// TIA Portal project "Industrial Oven Control" (V17)
// Industrial Oven Control
// The oven should preheat for 10s, then maintain the set temperature for 20 sec and then cool down for 30 sec.

(* hardware
DEVICE "S7-1200 station_1"  S7-1200 Station
   slot 0: "Rack_0"  S7-1200 Rack  Rack  V1.0
   slot 1: "PLC_1"  CPU 1215C AC/DC/Rly  6ES7 215-1BG40-0XB0  V4.5
*)

// ===== PLC "PLC_1"  CPU 1215C AC/DC/Rly =====

VAR_GLOBAL   // PLC tag table "Default tag table"
   "Turn_ON" AT %I0.0 : Bool;
   "Pre-Heat" AT %Q0.0 : Bool;
   "Set Temp" AT %Q0.1 : Bool;
   "Cooling" AT %Q0.2 : Bool;
END_VAR

// folder: System blocks/Program resources

DATA_BLOCK "IEC_Timer_0_DB"   // DB1
{ S7_Optimized_Access := 'TRUE' }
AUTHOR : Simatic
FAMILY : IEC
NAME : IEC_TMR
VERSION : 1.0
// stored: InstanceOfName IEC_TIMER
"IEC_TIMER"
BEGIN
END_DATA_BLOCK

DATA_BLOCK "IEC_Timer_0_DB_1"   // DB2
{ S7_Optimized_Access := 'TRUE' }
AUTHOR : Simatic
FAMILY : IEC
NAME : IEC_TMR
VERSION : 1.0
// stored: InstanceOfName IEC_TIMER
"IEC_TIMER"
BEGIN
END_DATA_BLOCK

DATA_BLOCK "IEC_Timer_0_DB_2"   // DB3
{ S7_Optimized_Access := 'TRUE' }
AUTHOR : Simatic
FAMILY : IEC
NAME : IEC_TMR
VERSION : 1.0
// stored: InstanceOfName IEC_TIMER
"IEC_TIMER"
BEGIN
END_DATA_BLOCK

DATA_BLOCK "IEC_Timer_0_DB_3"   // DB4
{ S7_Optimized_Access := 'TRUE' }
AUTHOR : Simatic
FAMILY : IEC
NAME : IEC_TMR
VERSION : 1.0
// stored: InstanceOfName IEC_TIMER
"IEC_TIMER"
BEGIN
END_DATA_BLOCK

DATA_BLOCK "IEC_Timer_0_DB_4"   // DB5
{ S7_Optimized_Access := 'TRUE' }
AUTHOR : Simatic
FAMILY : IEC
NAME : IEC_TMR
VERSION : 1.0
// stored: InstanceOfName IEC_TIMER
"IEC_TIMER"
BEGIN
END_DATA_BLOCK

// folder: (top level)

ORGANIZATION_BLOCK "Main"   // OB1, LAD, ProgramCycle
TITLE = "Main Program Sweep (Cycle)"
{ S7_Optimized_Access := 'TRUE' }
VERSION : 0.1
   VAR_INPUT
      Initial_Call : Bool;   // Initial call of this OB
      Remanence : Bool;   // =True, if remanent data are available
   END_VAR
BEGIN

REGION Network 1
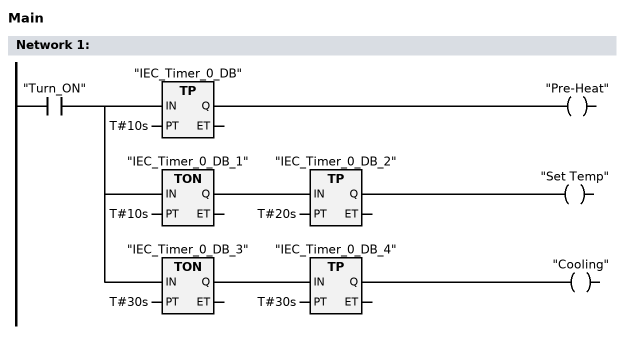
   "IEC_Timer_0_DB".TP(IN := "Turn_ON", PT := T#10s);
   "Pre-Heat" := "IEC_Timer_0_DB".Q;
   "IEC_Timer_0_DB_1".TON(IN := "Turn_ON", PT := T#10s);
   "IEC_Timer_0_DB_2".TP(IN := "IEC_Timer_0_DB_1".Q, PT := T#20s);
   "Set Temp" := "IEC_Timer_0_DB_2".Q;
   "IEC_Timer_0_DB_3".TON(IN := "Turn_ON", PT := T#30s);
   "IEC_Timer_0_DB_4".TP(IN := "IEC_Timer_0_DB_3".Q, PT := T#30s);
   "Cooling" := "IEC_Timer_0_DB_4".Q;
END_REGION
END_ORGANIZATION_BLOCK